{warning 'TODO: Example'}
//{error 'TODO: Example'}
PROGRAM MAIN
VAR	
	// Objects:
	eMainState : E_MainState := E_MainState.Initialization; //This enumeration handles the case statement in main
	fbModeHandler : FB_ModeHandler; //ModeHandler is where the end user states are handled
	fbTimestamp : FB_Timestamp; //Create a timestamp object
	fbDbEventLogger : FB_DbEventLogger;	
	
	// Event Log Variables:
	aMainEventLog : ARRAY[1..SystemConfig.MAIN_EVENT_LOG_MAX_LENGTH] OF ST_Event; // Error-log array
	nMainEventLogSize : UINT := 0; // The length of the array with valid errors
	nEventLogErrorCounter : ULINT := 0;	// Error tracking during logging. if this starts to accumulate, need to adjust buffer parameters in FB_DbEventLogger
	nEventCounter : ULINT := 0; // Number of events accumulated during run-time
	
	// Database FB Error Handling IO:
	bDbEnabled : BOOL := TRUE; // change to false to run local without DB
	bDbCriticalError : BOOL := FALSE;
	sDbCriticalErrorMessage : T_MaxString;
	bCaseEnded : BOOL := FALSE;
	
END_VAR

UpdateTimeStamps(); //Method from fbTimestamp object to update the current timestamp as of the PLC cycle
CheckEstopReset(); // TODO: Add this back in when ESTOP program is redone
CheckDbFailure();
		
CASE eMainState OF
	
	E_MainState.Initialization :
	
		IF bDbEnabled THEN
			IF NOT fbDbEventLogger.DbCreated THEN
				EventLogInit();
			ELSE
				Setup();
				eMainState := E_MainState.Running;
			END_IF
		ELSE
			Setup();
			eMainState := E_MainState.Running;
		END_IF
		

	E_MainState.Running :

		fbModeHandler();
		IF bDbEnabled THEN
			nEventCounter := nEventCounter + nMainEventLogSize; 
			LogPlcCycleEvents(); // Queue the current cycle's events before next cycle starts
		END_IF
		
		// Catch the end of a case
		IF fbModeHandler.InnerState = E_ModeHandlerStates.EndCase THEN
			bCaseEnded := TRUE;
		END_IF
		
		// Catch the transition from end-case to Idle before shutting down Database
		IF bCaseEnded AND (fbModeHandler.InnerState = E_ModeHandlerStates.Idle) THEN
			eMainState:= E_MainState.Shutdown;
			bCaseEnded := FALSE;
		END_IF
		
	E_MainState.Shutdown : 
		IF bDbEnabled THEN		
			IF EventLogClose() THEN
				EventLogReset();
				eMainState := E_MainState.Idle;
			END_IF
		ELSE
			eMainState := E_MainState.Idle;
		END_IF
		
	E_MainState.Idle:
		fbModeHandler(); // mode handler should be idle, no event logging necessary here, just polling for updates

		IF fbModeHandler.InnerState <> E_ModeHandlerStates.Idle THEN
			eMainState:= E_MainState.Initialization;
		END_IF
		
	E_MainState.DbFailure:
		// Failure mode, initialization failed, PLC program should not be allowed to continue.
		sDbCriticalErrorMessage := fbDbEventLogger.sCriticalErrorMessage;

END_CASE;

METHOD PRIVATE CheckDbFailure : BOOL
VAR_INPUT
END_VAR
sDbCriticalErrorMessage := fbDbEventLogger.sCriticalErrorMessage;
IF fbDbEventLogger.bCriticalError THEN
	bDbCriticalError := TRUE;
	eMainState := E_MainState.DbFailure;
END_IF
END_METHOD

METHOD CheckEstopReset : BOOL

IF Safety.GVL_bEstopErrACK THEN
	Safety.GVL_bEstopErrACK := FALSE;
	//Update Reset signal
//	Safety.GVL_bEstopReset := Safety.GVL_bEstopResetInput; // TODO: update safety program to have reset directly linked to EL1259 Channel8 input
	Safety.GVL_bEstopReset := TRUE;			
	Safety.GVL_bEstopRun := TRUE;
ELSE
	IF Safety.GVL_bEstopResetInput THEN
		Safety.GVL_bEstopRun := FALSE;
		Safety.GVL_bEstopErrACK := TRUE;
	ELSE
		Safety.GVL_bEstopReset := FALSE;
	END_IF

END_IF
END_METHOD

METHOD PRIVATE EventLogClose : BOOL
// Keep calling DbClosed Until finished
IF NOT fbDbEventLogger.DbClosed THEN
	fbDbEventLogger(bClose:=TRUE);
	EventLogClose:= FALSE;
ELSE
	EventLogClose:=TRUE;
END_IF
END_METHOD

METHOD PRIVATE EventLogInit : BOOL
fbDbEventLogger(sAmsNetId:=SystemConfig.AMS_NET_ID, 
					sDbPath:= SystemConfig.EVENT_LOG_DIR_PATH, 
							sTimestamp:=DateTime.GVL_DATE_STRING,
								stEventArrayIn:=aMainEventLog,
									nEventArraySize:=nMainEventLogSize);
END_METHOD

METHOD PRIVATE EventLogReset : BOOL
fbDbEventLogger(bResetDbInitialization := TRUE);
END_METHOD

METHOD PRIVATE LogPlcCycleEvents : BOOL
fbDbEventLogger(); // Buffer the current plc cycle's events
IF fbDbEventLogger.bError THEN
	nEventLogErrorCounter := nEventLogErrorCounter + 1; 
ELSE
	LogPlcCycleEvents := TRUE;
END_IF
END_METHOD

METHOD PRIVATE Setup : BOOL
fbModeHandler(eStateSourceID := E_StateSourceID.ModeHandler, 
						aErrorLog := aMainEventLog,
							 nErrorLogIndex := nMainEventLogSize);
END_METHOD

METHOD PRIVATE UpdateTimeStamps : BOOL
fbTimestamp.UpdateTimestamp();
DateTime.GVL_DATE_STRING := fbTimestamp.DateString;
DateTime.GVL_DATE_TIME := fbTimestamp.DateTime;
DateTime.GVL_TIME_STRING := fbTimestamp.TimeString;
END_METHOD

END_PROGRAM

(* stored: Version 1.1.0.1, ProductVersion 3.1.4024.12
   POU MAIN: Id {54cdbe1a-8209-49db-bd38-4bf5a679b4fd}, SpecialFunc None
   Method CheckDbFailure: Id {b0f6aa1a-80c6-429b-8bbc-da4c2bcfb131}
   Method CheckEstopReset: Id {73a2a8dd-d948-4e7f-bebf-9e865babfe6f}
   Method EventLogClose: Id {ba1a6545-8c1b-4e79-89c7-e5ba34d7ef7c}
   Method EventLogInit: Id {e9404fa5-32bc-4830-b1ec-8f1e2a960b48}
   Method EventLogReset: Id {fa2b3b9e-aa52-4440-9ac1-98635225456d}
   Method LogPlcCycleEvents: Id {cab6421a-2909-4dc7-8cfc-fa6ced084c02}
   Method Setup: Id {8798fdf3-47bd-4fa4-b448-3179e9ef5d3c}
   Method UpdateTimeStamps: Id {ecd72610-919d-4e3a-9cd2-e9d635f68cde} *)
